PROGRAM POU_1
VAR
	tCzas: TIME := T#3S;
	TON1: TON;
	TON2: TON;
END_VAR

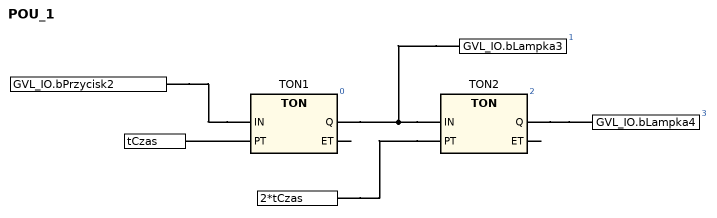
TON1(IN := GVL_IO.bPrzycisk2, PT := tCzas); // TON
GVL_IO.bLampka3 := TON1.Q;
TON2(IN := TON1.Q, PT := 2*tCzas); // TON
GVL_IO.bLampka4 := TON2.Q;

END_PROGRAM

(* stored: Version 1.1.0.1, ProductVersion 3.1.4024.12
   POU POU_1: Id {11ffe61b-f5d4-4811-a885-ad88d7a3bc48}, SpecialFunc None *)
